{attribute 'qualified_only'}
VAR_GLOBAL
	stFromMCToOC AT %I* : FromMainControlToOperationControl;
	stFromOCToMC AT %Q* : FromOperationControlToMainControl;
	
	iTest AT %I* : INT;
END_VAR

(* stored: Version 1.1.0.1, ProductVersion 3.1.4024.12
   GVL GVL: Id {6a7924c9-ad45-4856-a589-50627d8de83c} *)
